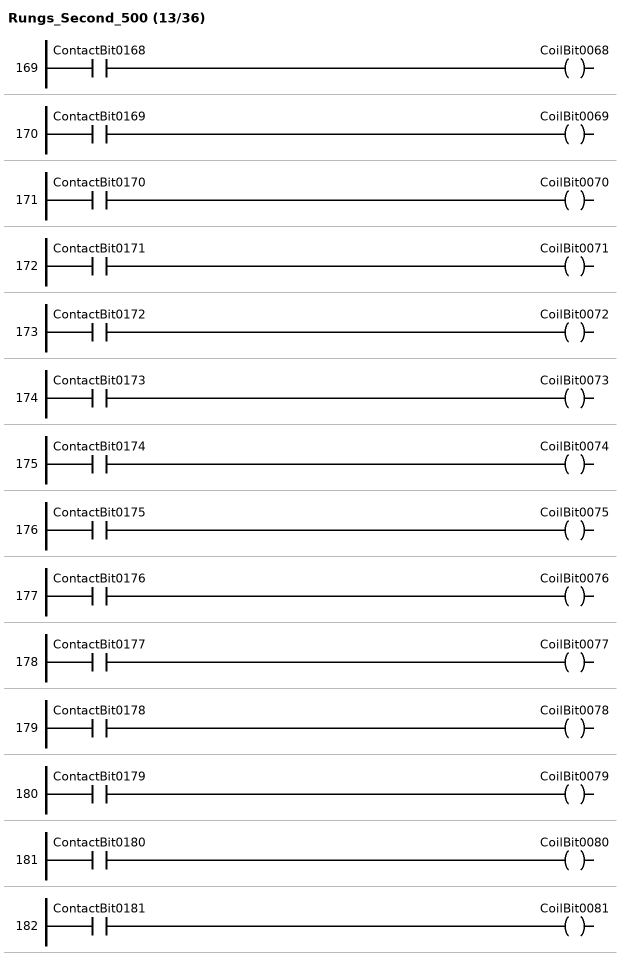
// NETWORK 169
CoilBit0068 := ContactBit0168;

// NETWORK 170
CoilBit0069 := ContactBit0169;

// NETWORK 171
CoilBit0070 := ContactBit0170;

// NETWORK 172
CoilBit0071 := ContactBit0171;

// NETWORK 173
CoilBit0072 := ContactBit0172;

// NETWORK 174
CoilBit0073 := ContactBit0173;

// NETWORK 175
CoilBit0074 := ContactBit0174;

// NETWORK 176
CoilBit0075 := ContactBit0175;

// NETWORK 177
CoilBit0076 := ContactBit0176;

// NETWORK 178
CoilBit0077 := ContactBit0177;

// NETWORK 179
CoilBit0078 := ContactBit0178;

// NETWORK 180
CoilBit0079 := ContactBit0179;

// NETWORK 181
CoilBit0080 := ContactBit0180;

// NETWORK 182
CoilBit0081 := ContactBit0181;

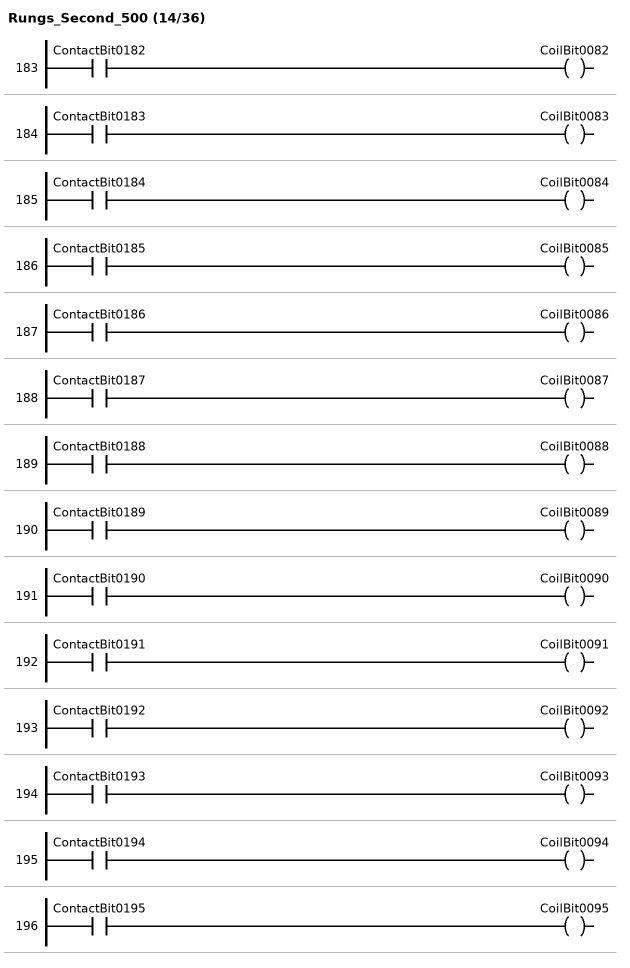
// NETWORK 183
CoilBit0082 := ContactBit0182;

// NETWORK 184
CoilBit0083 := ContactBit0183;

// NETWORK 185
CoilBit0084 := ContactBit0184;

// NETWORK 186
CoilBit0085 := ContactBit0185;

// NETWORK 187
CoilBit0086 := ContactBit0186;

// NETWORK 188
CoilBit0087 := ContactBit0187;

// NETWORK 189
CoilBit0088 := ContactBit0188;

// NETWORK 190
CoilBit0089 := ContactBit0189;

// NETWORK 191
CoilBit0090 := ContactBit0190;

// NETWORK 192
CoilBit0091 := ContactBit0191;

// NETWORK 193
CoilBit0092 := ContactBit0192;

// NETWORK 194
CoilBit0093 := ContactBit0193;

// NETWORK 195
CoilBit0094 := ContactBit0194;

// NETWORK 196
CoilBit0095 := ContactBit0195;

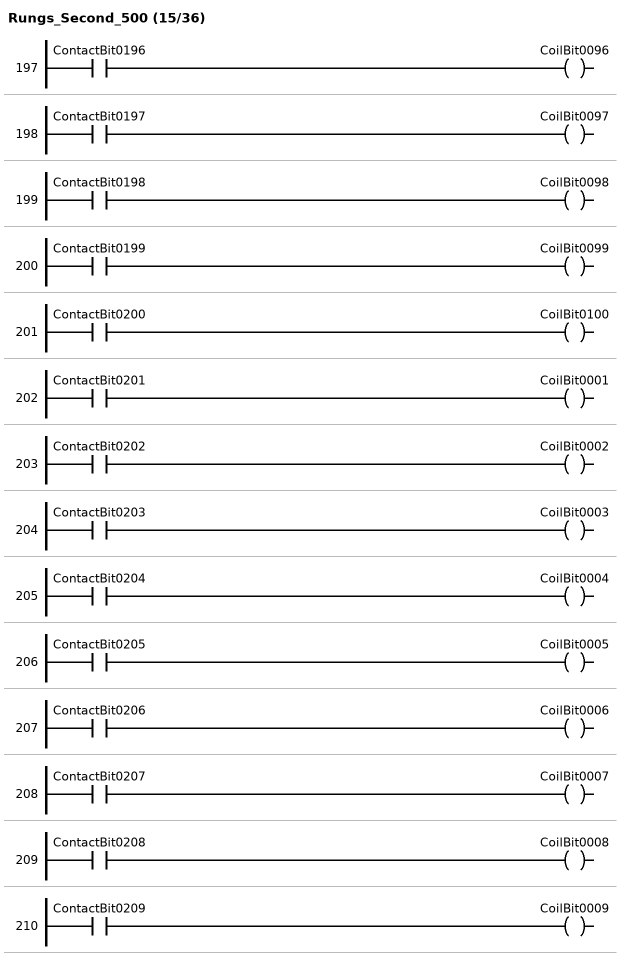
// NETWORK 197
CoilBit0096 := ContactBit0196;

// NETWORK 198
CoilBit0097 := ContactBit0197;

// NETWORK 199
CoilBit0098 := ContactBit0198;

// NETWORK 200
CoilBit0099 := ContactBit0199;

// NETWORK 201
CoilBit0100 := ContactBit0200;

// NETWORK 202
CoilBit0001 := ContactBit0201;

// NETWORK 203
CoilBit0002 := ContactBit0202;

// NETWORK 204
CoilBit0003 := ContactBit0203;

// NETWORK 205
CoilBit0004 := ContactBit0204;

// NETWORK 206
CoilBit0005 := ContactBit0205;

// NETWORK 207
CoilBit0006 := ContactBit0206;

// NETWORK 208
CoilBit0007 := ContactBit0207;

// NETWORK 209
CoilBit0008 := ContactBit0208;

// NETWORK 210
CoilBit0009 := ContactBit0209;

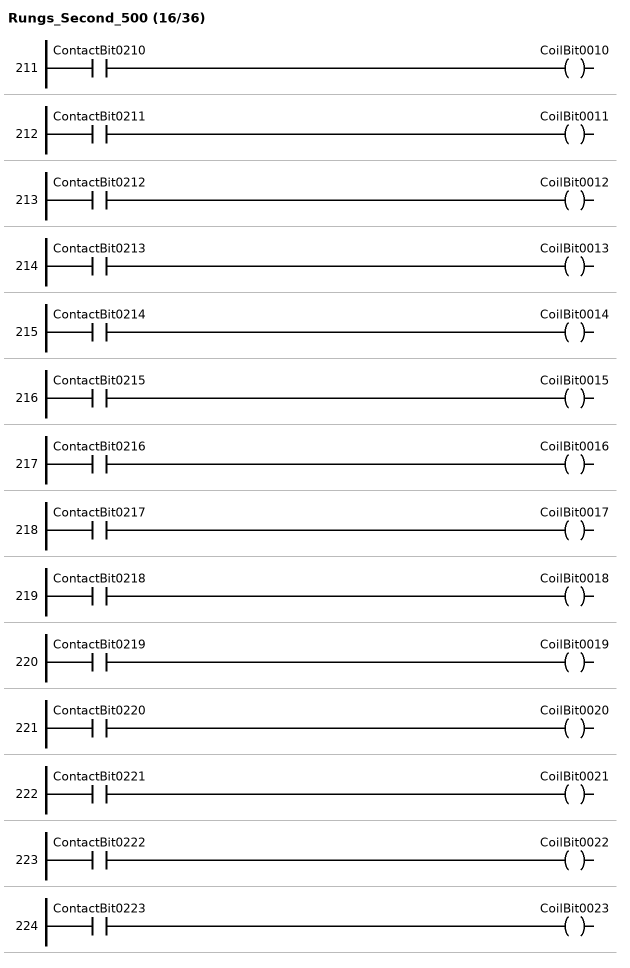
// NETWORK 211
CoilBit0010 := ContactBit0210;

// NETWORK 212
CoilBit0011 := ContactBit0211;

// NETWORK 213
CoilBit0012 := ContactBit0212;

// NETWORK 214
CoilBit0013 := ContactBit0213;

// NETWORK 215
CoilBit0014 := ContactBit0214;

// NETWORK 216
CoilBit0015 := ContactBit0215;

// NETWORK 217
CoilBit0016 := ContactBit0216;

// NETWORK 218
CoilBit0017 := ContactBit0217;

// NETWORK 219
CoilBit0018 := ContactBit0218;

// NETWORK 220
CoilBit0019 := ContactBit0219;

// NETWORK 221
CoilBit0020 := ContactBit0220;

// NETWORK 222
CoilBit0021 := ContactBit0221;

// NETWORK 223
CoilBit0022 := ContactBit0222;

// NETWORK 224
CoilBit0023 := ContactBit0223;

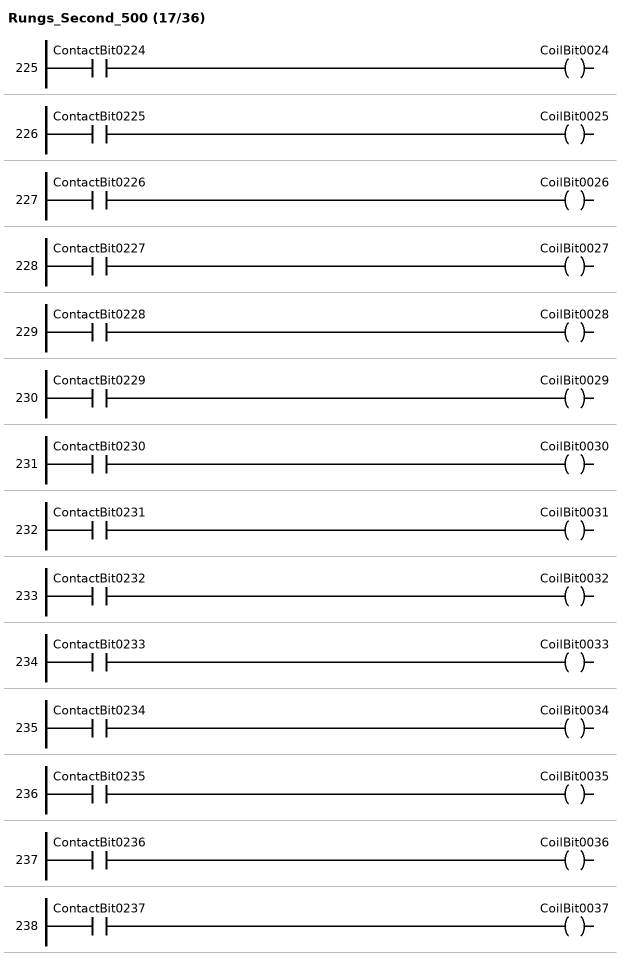
// NETWORK 225
CoilBit0024 := ContactBit0224;

// NETWORK 226
CoilBit0025 := ContactBit0225;

// NETWORK 227
CoilBit0026 := ContactBit0226;

// NETWORK 228
CoilBit0027 := ContactBit0227;

// NETWORK 229
CoilBit0028 := ContactBit0228;

// NETWORK 230
CoilBit0029 := ContactBit0229;

// NETWORK 231
CoilBit0030 := ContactBit0230;

// NETWORK 232
CoilBit0031 := ContactBit0231;

// NETWORK 233
CoilBit0032 := ContactBit0232;

// NETWORK 234
CoilBit0033 := ContactBit0233;

// NETWORK 235
CoilBit0034 := ContactBit0234;

// NETWORK 236
CoilBit0035 := ContactBit0235;

// NETWORK 237
CoilBit0036 := ContactBit0236;

// NETWORK 238
CoilBit0037 := ContactBit0237;

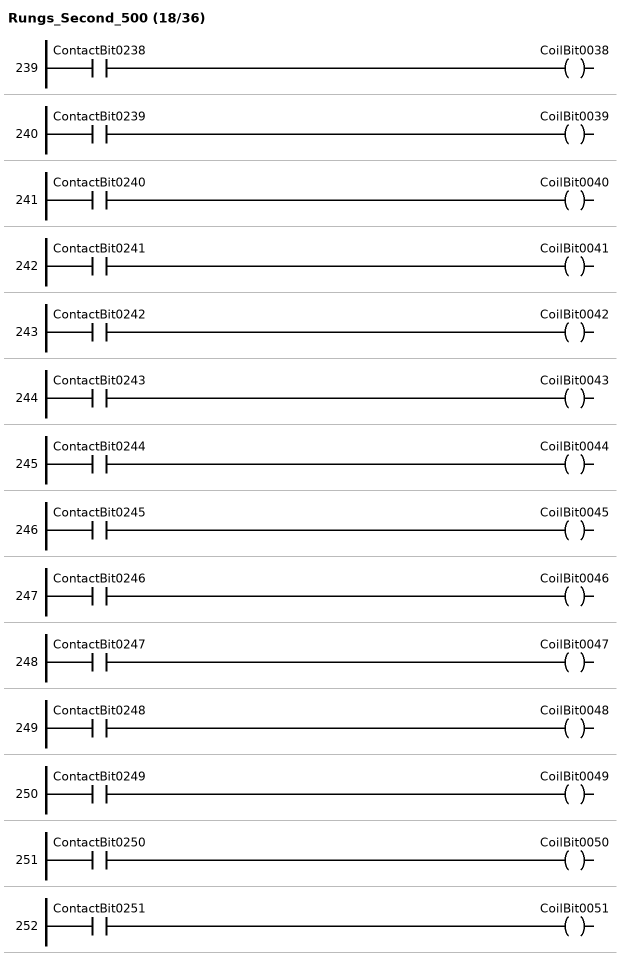
// NETWORK 239
CoilBit0038 := ContactBit0238;

// NETWORK 240
CoilBit0039 := ContactBit0239;

// NETWORK 241
CoilBit0040 := ContactBit0240;

// NETWORK 242
CoilBit0041 := ContactBit0241;

// NETWORK 243
CoilBit0042 := ContactBit0242;

// NETWORK 244
CoilBit0043 := ContactBit0243;

// NETWORK 245
CoilBit0044 := ContactBit0244;

// NETWORK 246
CoilBit0045 := ContactBit0245;

// NETWORK 247
CoilBit0046 := ContactBit0246;

// NETWORK 248
CoilBit0047 := ContactBit0247;

// NETWORK 249
CoilBit0048 := ContactBit0248;

// NETWORK 250
CoilBit0049 := ContactBit0249;

// NETWORK 251
CoilBit0050 := ContactBit0250;

// NETWORK 252
CoilBit0051 := ContactBit0251;

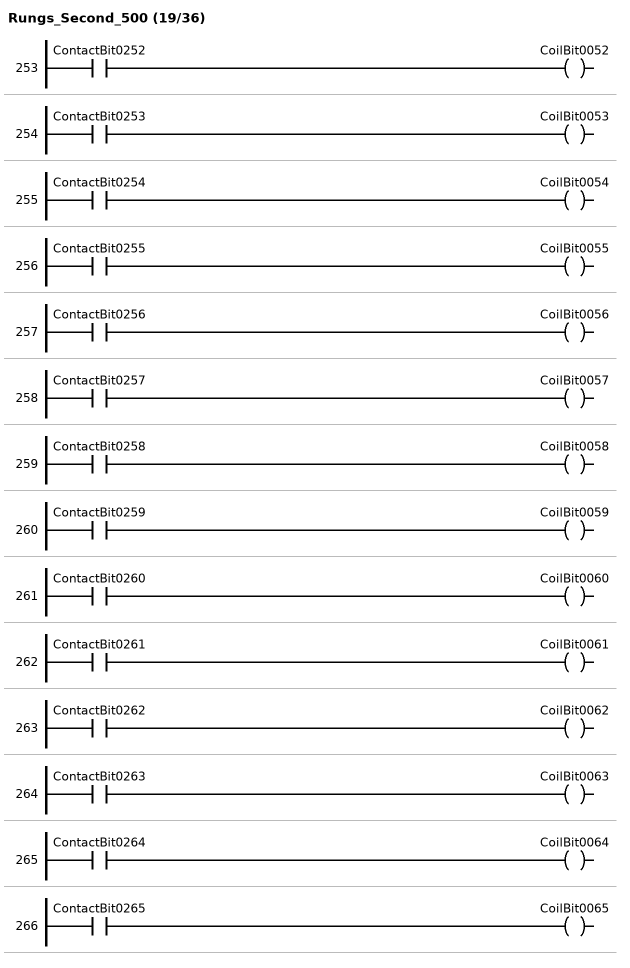
// NETWORK 253
CoilBit0052 := ContactBit0252;

// NETWORK 254
CoilBit0053 := ContactBit0253;

// NETWORK 255
CoilBit0054 := ContactBit0254;

// NETWORK 256
CoilBit0055 := ContactBit0255;

// NETWORK 257
CoilBit0056 := ContactBit0256;

// NETWORK 258
CoilBit0057 := ContactBit0257;

// NETWORK 259
CoilBit0058 := ContactBit0258;

// NETWORK 260
CoilBit0059 := ContactBit0259;

// NETWORK 261
CoilBit0060 := ContactBit0260;

// NETWORK 262
CoilBit0061 := ContactBit0261;

// NETWORK 263
CoilBit0062 := ContactBit0262;

// NETWORK 264
CoilBit0063 := ContactBit0263;

// NETWORK 265
CoilBit0064 := ContactBit0264;

// NETWORK 266
CoilBit0065 := ContactBit0265;

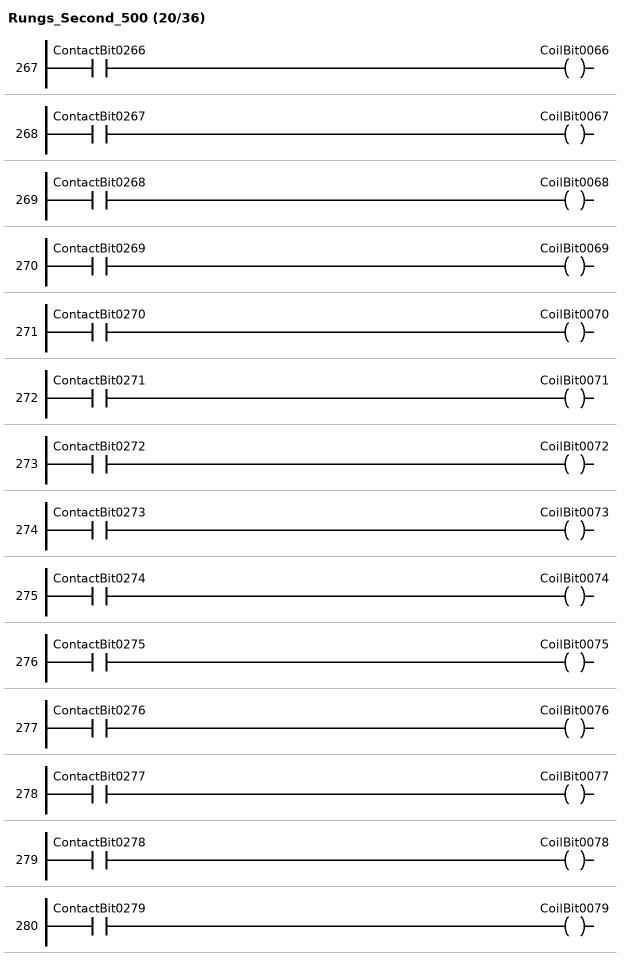
// NETWORK 267
CoilBit0066 := ContactBit0266;

// NETWORK 268
CoilBit0067 := ContactBit0267;

// NETWORK 269
CoilBit0068 := ContactBit0268;

// NETWORK 270
CoilBit0069 := ContactBit0269;

// NETWORK 271
CoilBit0070 := ContactBit0270;

// NETWORK 272
CoilBit0071 := ContactBit0271;

// NETWORK 273
CoilBit0072 := ContactBit0272;

// NETWORK 274
CoilBit0073 := ContactBit0273;

// NETWORK 275
CoilBit0074 := ContactBit0274;

// NETWORK 276
CoilBit0075 := ContactBit0275;

// NETWORK 277
CoilBit0076 := ContactBit0276;

// NETWORK 278
CoilBit0077 := ContactBit0277;

// NETWORK 279
CoilBit0078 := ContactBit0278;

// NETWORK 280
CoilBit0079 := ContactBit0279;

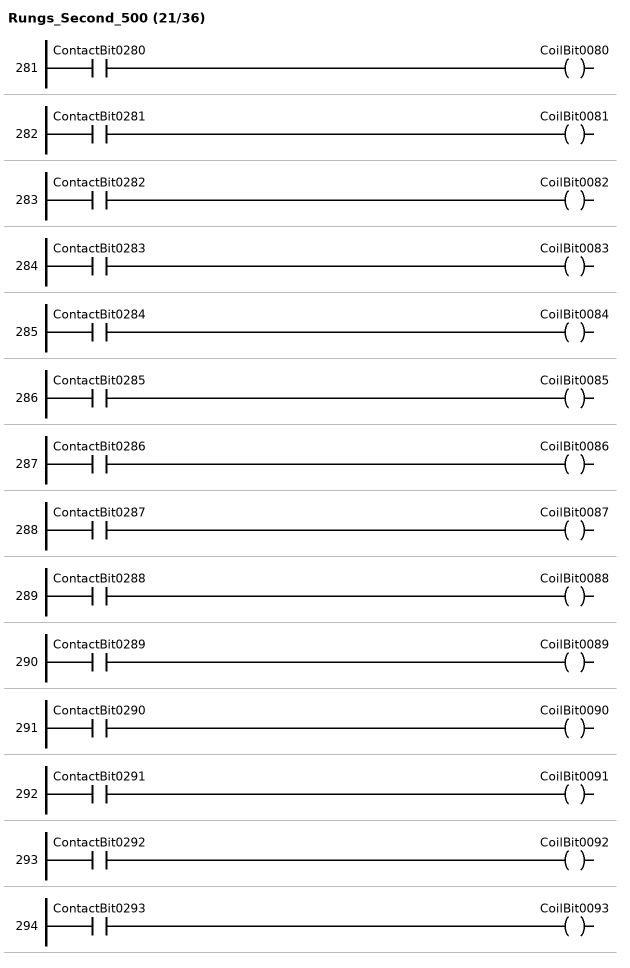
// NETWORK 281
CoilBit0080 := ContactBit0280;

// NETWORK 282
CoilBit0081 := ContactBit0281;

// NETWORK 283
CoilBit0082 := ContactBit0282;

// NETWORK 284
CoilBit0083 := ContactBit0283;

// NETWORK 285
CoilBit0084 := ContactBit0284;

// NETWORK 286
CoilBit0085 := ContactBit0285;

// NETWORK 287
CoilBit0086 := ContactBit0286;

// NETWORK 288
CoilBit0087 := ContactBit0287;

// NETWORK 289
CoilBit0088 := ContactBit0288;

// NETWORK 290
CoilBit0089 := ContactBit0289;

// NETWORK 291
CoilBit0090 := ContactBit0290;

// NETWORK 292
CoilBit0091 := ContactBit0291;

// NETWORK 293
CoilBit0092 := ContactBit0292;

// NETWORK 294
CoilBit0093 := ContactBit0293;

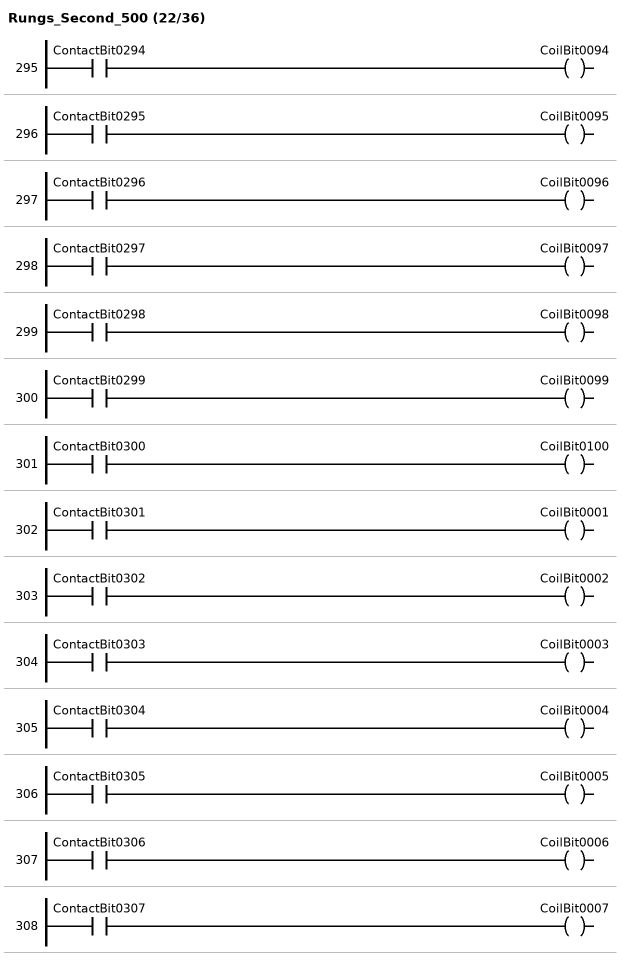
// NETWORK 295
CoilBit0094 := ContactBit0294;

// NETWORK 296
CoilBit0095 := ContactBit0295;

// NETWORK 297
CoilBit0096 := ContactBit0296;

// NETWORK 298
CoilBit0097 := ContactBit0297;

// NETWORK 299
CoilBit0098 := ContactBit0298;

// NETWORK 300
CoilBit0099 := ContactBit0299;

// NETWORK 301
CoilBit0100 := ContactBit0300;

// NETWORK 302
CoilBit0001 := ContactBit0301;

// NETWORK 303
CoilBit0002 := ContactBit0302;

// NETWORK 304
CoilBit0003 := ContactBit0303;

// NETWORK 305
CoilBit0004 := ContactBit0304;

// NETWORK 306
CoilBit0005 := ContactBit0305;

// NETWORK 307
CoilBit0006 := ContactBit0306;

// NETWORK 308
CoilBit0007 := ContactBit0307;

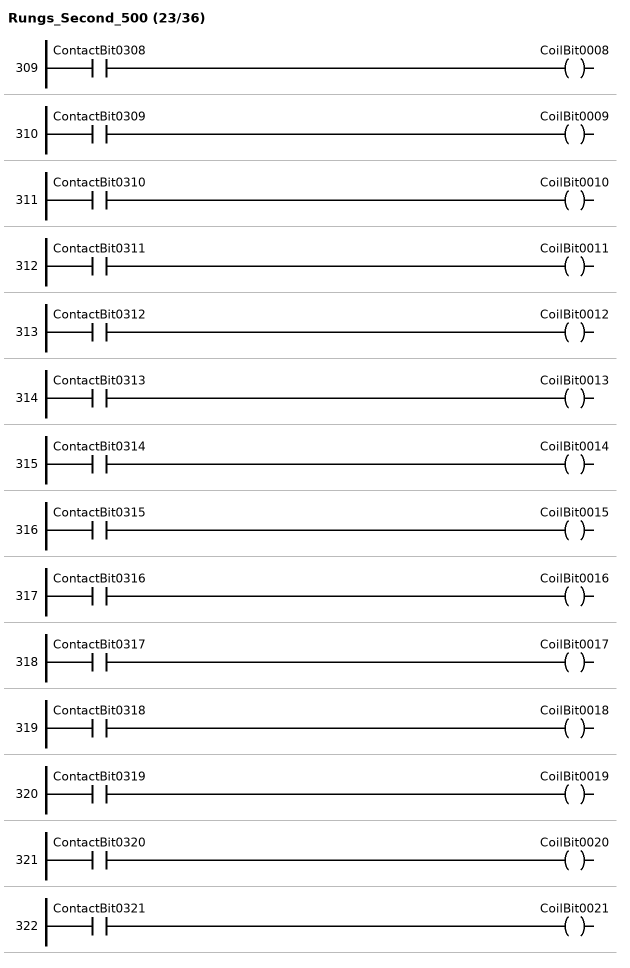
// NETWORK 309
CoilBit0008 := ContactBit0308;

// NETWORK 310
CoilBit0009 := ContactBit0309;

// NETWORK 311
CoilBit0010 := ContactBit0310;

// NETWORK 312
CoilBit0011 := ContactBit0311;

// NETWORK 313
CoilBit0012 := ContactBit0312;

// NETWORK 314
CoilBit0013 := ContactBit0313;

// NETWORK 315
CoilBit0014 := ContactBit0314;

// NETWORK 316
CoilBit0015 := ContactBit0315;

// NETWORK 317
CoilBit0016 := ContactBit0316;

// NETWORK 318
CoilBit0017 := ContactBit0317;

// NETWORK 319
CoilBit0018 := ContactBit0318;

// NETWORK 320
CoilBit0019 := ContactBit0319;

// NETWORK 321
CoilBit0020 := ContactBit0320;

// NETWORK 322
CoilBit0021 := ContactBit0321;

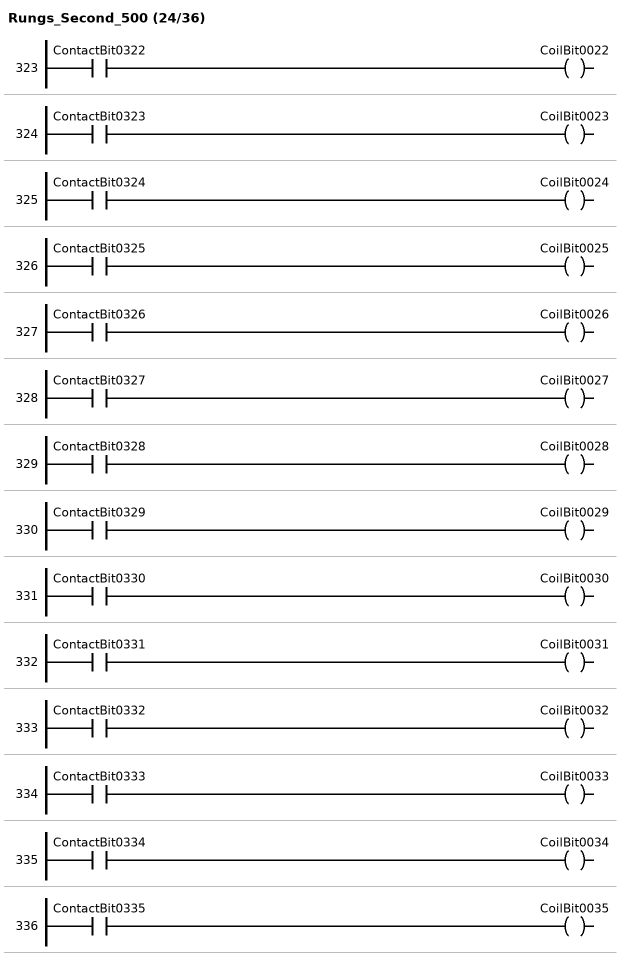
// NETWORK 323
CoilBit0022 := ContactBit0322;

// NETWORK 324
CoilBit0023 := ContactBit0323;

// NETWORK 325
CoilBit0024 := ContactBit0324;

// NETWORK 326
CoilBit0025 := ContactBit0325;

// NETWORK 327
CoilBit0026 := ContactBit0326;

// NETWORK 328
CoilBit0027 := ContactBit0327;

// NETWORK 329
CoilBit0028 := ContactBit0328;

// NETWORK 330
CoilBit0029 := ContactBit0329;

// NETWORK 331
CoilBit0030 := ContactBit0330;

// NETWORK 332
CoilBit0031 := ContactBit0331;

// NETWORK 333
CoilBit0032 := ContactBit0332;

// NETWORK 334
CoilBit0033 := ContactBit0333;

// NETWORK 335
CoilBit0034 := ContactBit0334;

// NETWORK 336
CoilBit0035 := ContactBit0335;

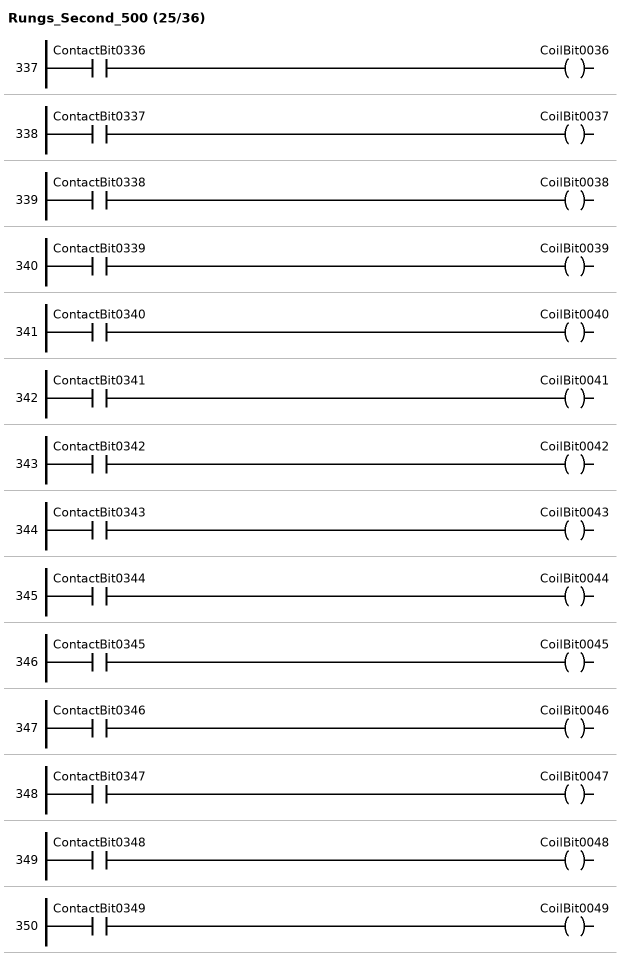
// NETWORK 337
CoilBit0036 := ContactBit0336;

// NETWORK 338
CoilBit0037 := ContactBit0337;

// NETWORK 339
CoilBit0038 := ContactBit0338;

// NETWORK 340
CoilBit0039 := ContactBit0339;

// NETWORK 341
CoilBit0040 := ContactBit0340;

// NETWORK 342
CoilBit0041 := ContactBit0341;

// NETWORK 343
CoilBit0042 := ContactBit0342;

// NETWORK 344
CoilBit0043 := ContactBit0343;

// NETWORK 345
CoilBit0044 := ContactBit0344;

// NETWORK 346
CoilBit0045 := ContactBit0345;

// NETWORK 347
CoilBit0046 := ContactBit0346;

// NETWORK 348
CoilBit0047 := ContactBit0347;

// NETWORK 349
CoilBit0048 := ContactBit0348;

// NETWORK 350
CoilBit0049 := ContactBit0349;

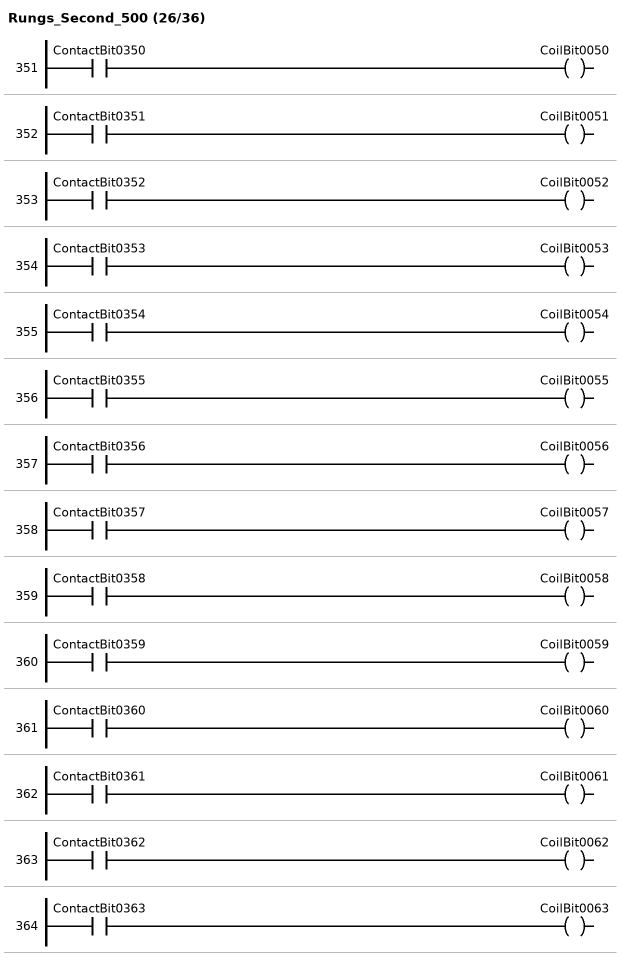
// NETWORK 351
CoilBit0050 := ContactBit0350;

// NETWORK 352
CoilBit0051 := ContactBit0351;

// NETWORK 353
CoilBit0052 := ContactBit0352;

// NETWORK 354
CoilBit0053 := ContactBit0353;

// NETWORK 355
CoilBit0054 := ContactBit0354;

// NETWORK 356
CoilBit0055 := ContactBit0355;

// NETWORK 357
CoilBit0056 := ContactBit0356;

// NETWORK 358
CoilBit0057 := ContactBit0357;

// NETWORK 359
CoilBit0058 := ContactBit0358;

// NETWORK 360
CoilBit0059 := ContactBit0359;

// NETWORK 361
CoilBit0060 := ContactBit0360;

// NETWORK 362
CoilBit0061 := ContactBit0361;

// NETWORK 363
CoilBit0062 := ContactBit0362;

// NETWORK 364
CoilBit0063 := ContactBit0363;

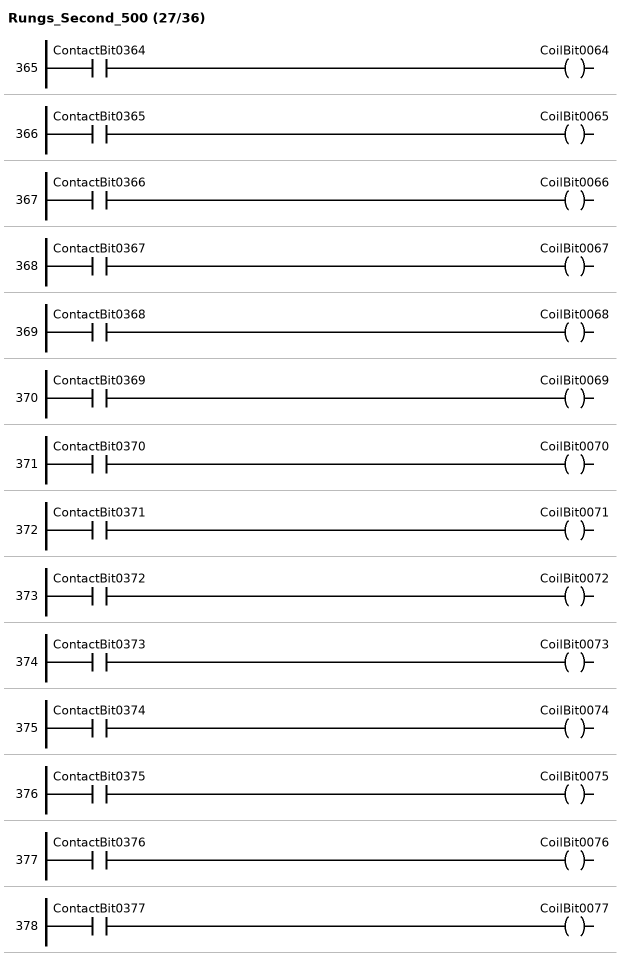
// NETWORK 365
CoilBit0064 := ContactBit0364;

// NETWORK 366
CoilBit0065 := ContactBit0365;

// NETWORK 367
CoilBit0066 := ContactBit0366;

// NETWORK 368
CoilBit0067 := ContactBit0367;

// NETWORK 369
CoilBit0068 := ContactBit0368;

// NETWORK 370
CoilBit0069 := ContactBit0369;

// NETWORK 371
CoilBit0070 := ContactBit0370;

// NETWORK 372
CoilBit0071 := ContactBit0371;

// NETWORK 373
CoilBit0072 := ContactBit0372;

// NETWORK 374
CoilBit0073 := ContactBit0373;

// NETWORK 375
CoilBit0074 := ContactBit0374;

// NETWORK 376
CoilBit0075 := ContactBit0375;

// NETWORK 377
CoilBit0076 := ContactBit0376;

// NETWORK 378
CoilBit0077 := ContactBit0377;

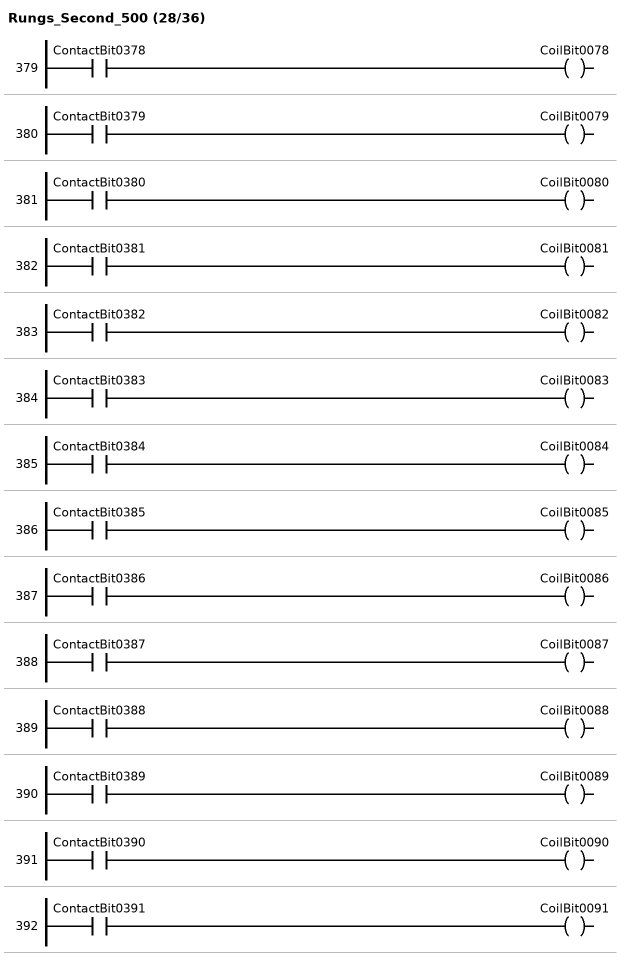
// NETWORK 379
CoilBit0078 := ContactBit0378;

// NETWORK 380
CoilBit0079 := ContactBit0379;

// NETWORK 381
CoilBit0080 := ContactBit0380;

// NETWORK 382
CoilBit0081 := ContactBit0381;

// NETWORK 383
CoilBit0082 := ContactBit0382;

// NETWORK 384
CoilBit0083 := ContactBit0383;

// NETWORK 385
CoilBit0084 := ContactBit0384;

// NETWORK 386
CoilBit0085 := ContactBit0385;

// NETWORK 387
CoilBit0086 := ContactBit0386;

// NETWORK 388
CoilBit0087 := ContactBit0387;

// NETWORK 389
CoilBit0088 := ContactBit0388;

// NETWORK 390
CoilBit0089 := ContactBit0389;

// NETWORK 391
CoilBit0090 := ContactBit0390;

// NETWORK 392
CoilBit0091 := ContactBit0391;

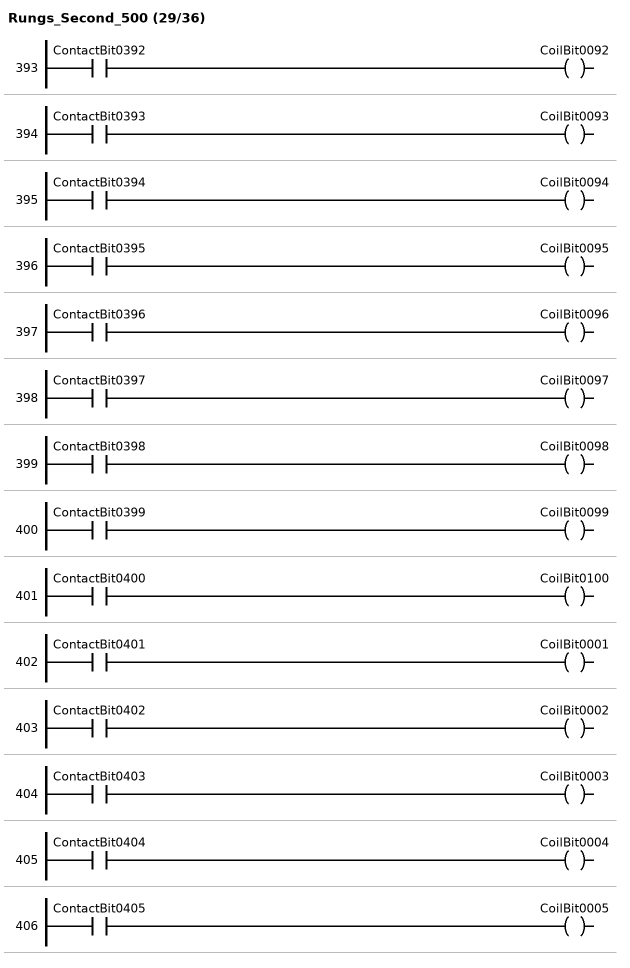
// NETWORK 393
CoilBit0092 := ContactBit0392;

// NETWORK 394
CoilBit0093 := ContactBit0393;

// NETWORK 395
CoilBit0094 := ContactBit0394;

// NETWORK 396
CoilBit0095 := ContactBit0395;

// NETWORK 397
CoilBit0096 := ContactBit0396;

// NETWORK 398
CoilBit0097 := ContactBit0397;

// NETWORK 399
CoilBit0098 := ContactBit0398;

// NETWORK 400
CoilBit0099 := ContactBit0399;

// NETWORK 401
CoilBit0100 := ContactBit0400;

// NETWORK 402
CoilBit0001 := ContactBit0401;

// NETWORK 403
CoilBit0002 := ContactBit0402;

// NETWORK 404
CoilBit0003 := ContactBit0403;

// NETWORK 405
CoilBit0004 := ContactBit0404;

// NETWORK 406
CoilBit0005 := ContactBit0405;

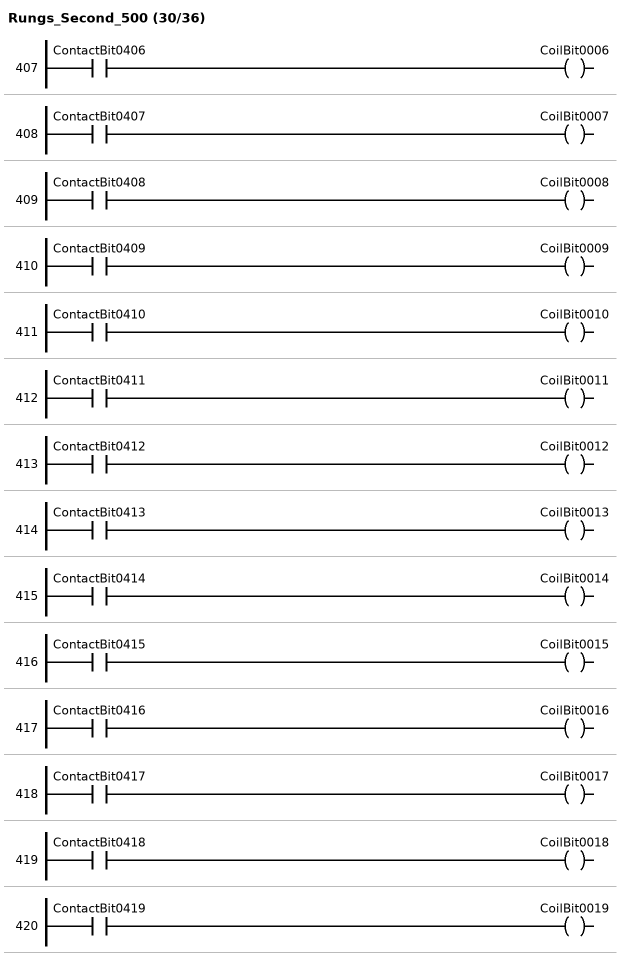
// NETWORK 407
CoilBit0006 := ContactBit0406;

// NETWORK 408
CoilBit0007 := ContactBit0407;

// NETWORK 409
CoilBit0008 := ContactBit0408;

// NETWORK 410
CoilBit0009 := ContactBit0409;

// NETWORK 411
CoilBit0010 := ContactBit0410;

// NETWORK 412
CoilBit0011 := ContactBit0411;

// NETWORK 413
CoilBit0012 := ContactBit0412;

// NETWORK 414
CoilBit0013 := ContactBit0413;

// NETWORK 415
CoilBit0014 := ContactBit0414;

// NETWORK 416
CoilBit0015 := ContactBit0415;

// NETWORK 417
CoilBit0016 := ContactBit0416;

// NETWORK 418
CoilBit0017 := ContactBit0417;

// NETWORK 419
CoilBit0018 := ContactBit0418;

// NETWORK 420
CoilBit0019 := ContactBit0419;

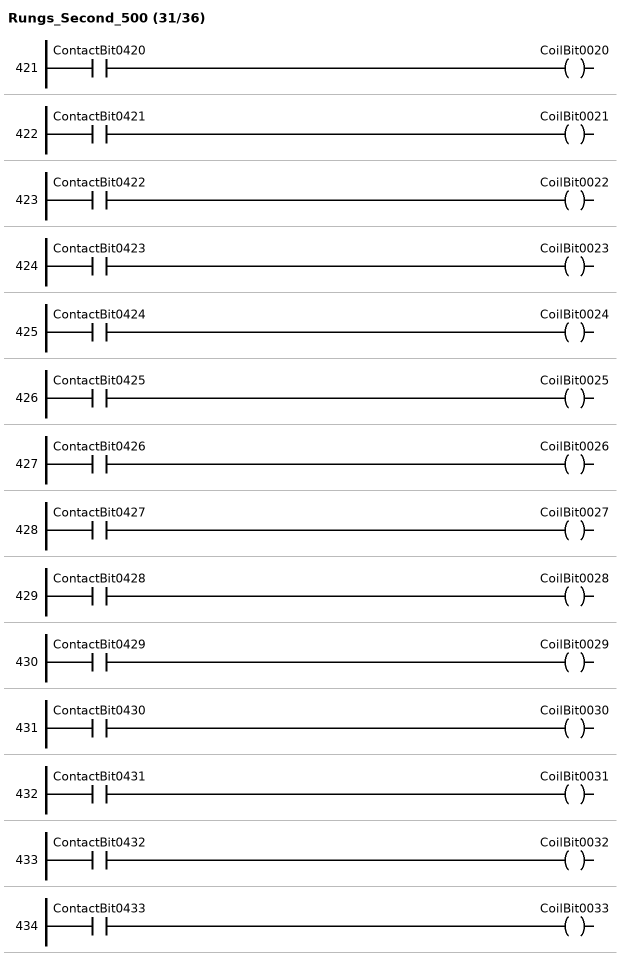
// NETWORK 421
CoilBit0020 := ContactBit0420;

// NETWORK 422
CoilBit0021 := ContactBit0421;

// NETWORK 423
CoilBit0022 := ContactBit0422;

// NETWORK 424
CoilBit0023 := ContactBit0423;

// NETWORK 425
CoilBit0024 := ContactBit0424;

// NETWORK 426
CoilBit0025 := ContactBit0425;

// NETWORK 427
CoilBit0026 := ContactBit0426;

// NETWORK 428
CoilBit0027 := ContactBit0427;

// NETWORK 429
CoilBit0028 := ContactBit0428;

// NETWORK 430
CoilBit0029 := ContactBit0429;

// NETWORK 431
CoilBit0030 := ContactBit0430;

// NETWORK 432
CoilBit0031 := ContactBit0431;

// NETWORK 433
CoilBit0032 := ContactBit0432;

// NETWORK 434
CoilBit0033 := ContactBit0433;

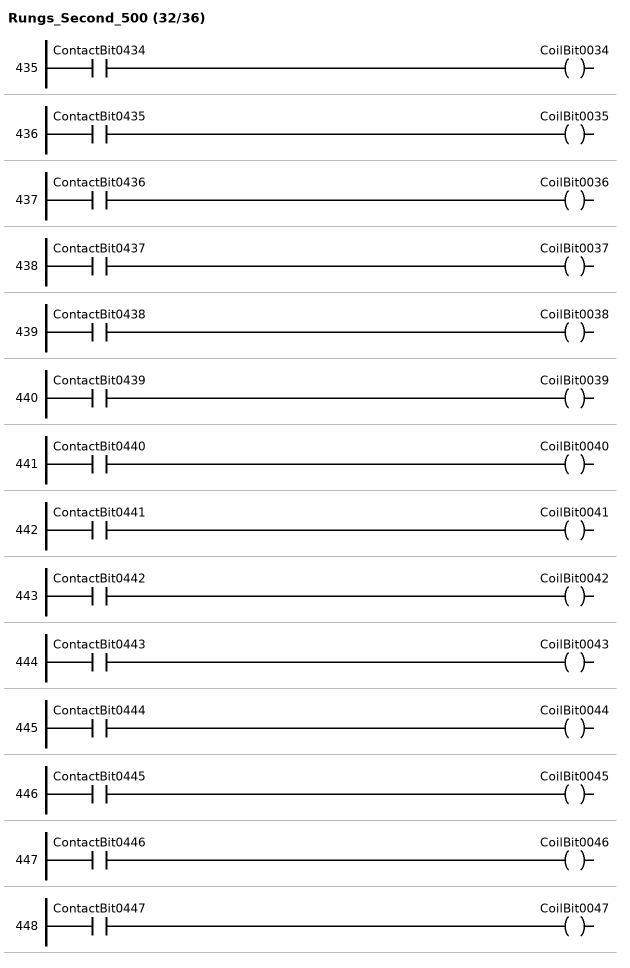
// NETWORK 435
CoilBit0034 := ContactBit0434;

// NETWORK 436
CoilBit0035 := ContactBit0435;

// NETWORK 437
CoilBit0036 := ContactBit0436;

// NETWORK 438
CoilBit0037 := ContactBit0437;

// NETWORK 439
CoilBit0038 := ContactBit0438;

// NETWORK 440
CoilBit0039 := ContactBit0439;

// NETWORK 441
CoilBit0040 := ContactBit0440;

// NETWORK 442
CoilBit0041 := ContactBit0441;

// NETWORK 443
CoilBit0042 := ContactBit0442;

// NETWORK 444
CoilBit0043 := ContactBit0443;

// NETWORK 445
CoilBit0044 := ContactBit0444;

// NETWORK 446
CoilBit0045 := ContactBit0445;

// NETWORK 447
CoilBit0046 := ContactBit0446;

// NETWORK 448
CoilBit0047 := ContactBit0447;

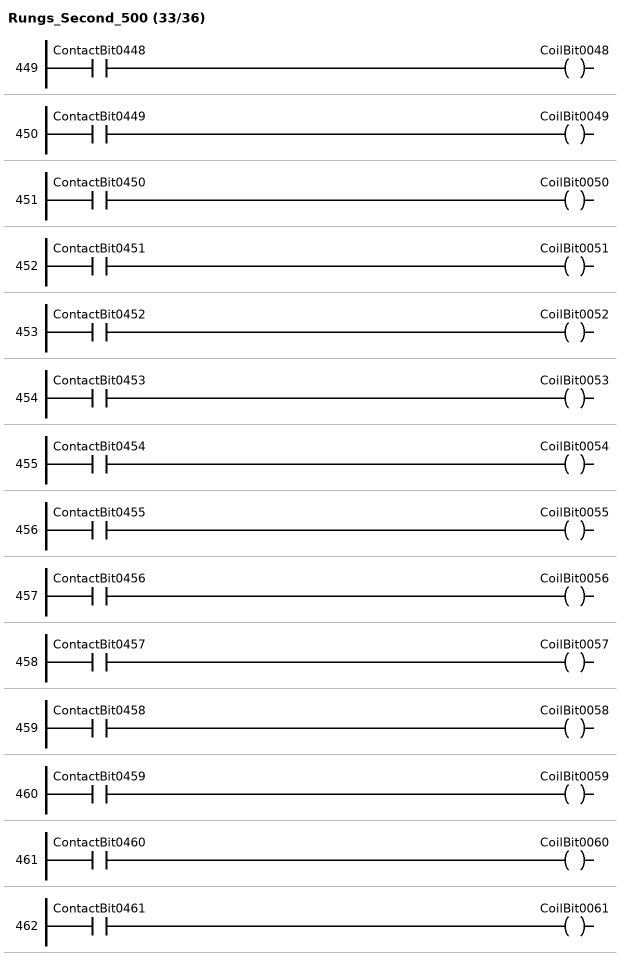
// NETWORK 449
CoilBit0048 := ContactBit0448;

// NETWORK 450
CoilBit0049 := ContactBit0449;

// NETWORK 451
CoilBit0050 := ContactBit0450;

// NETWORK 452
CoilBit0051 := ContactBit0451;

// NETWORK 453
CoilBit0052 := ContactBit0452;

// NETWORK 454
CoilBit0053 := ContactBit0453;

// NETWORK 455
CoilBit0054 := ContactBit0454;

// NETWORK 456
CoilBit0055 := ContactBit0455;

// NETWORK 457
CoilBit0056 := ContactBit0456;

// NETWORK 458
CoilBit0057 := ContactBit0457;

// NETWORK 459
CoilBit0058 := ContactBit0458;

// NETWORK 460
CoilBit0059 := ContactBit0459;

// NETWORK 461
CoilBit0060 := ContactBit0460;

// NETWORK 462
CoilBit0061 := ContactBit0461;

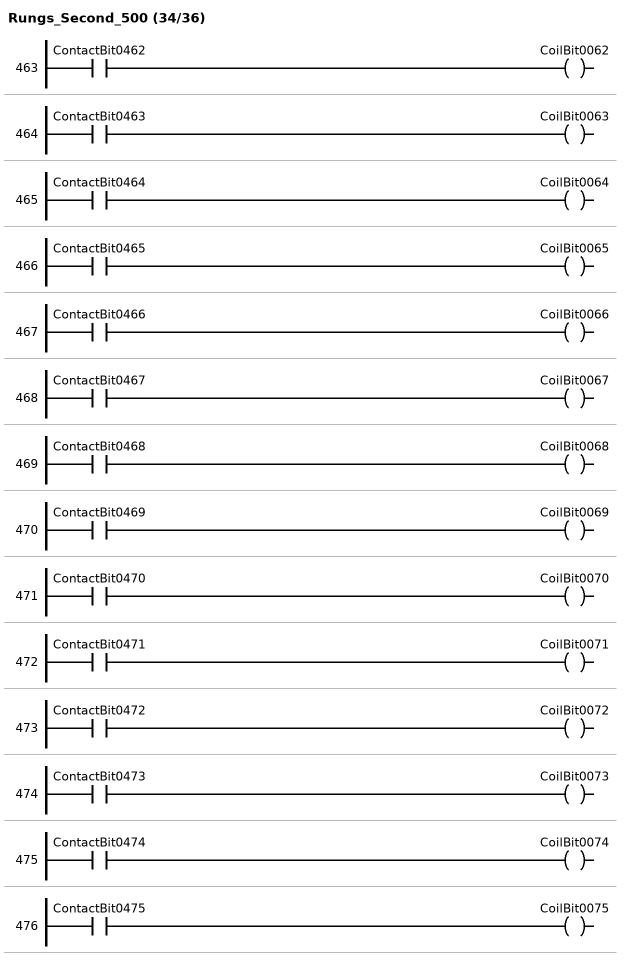
// NETWORK 463
CoilBit0062 := ContactBit0462;

// NETWORK 464
CoilBit0063 := ContactBit0463;

// NETWORK 465
CoilBit0064 := ContactBit0464;

// NETWORK 466
CoilBit0065 := ContactBit0465;

// NETWORK 467
CoilBit0066 := ContactBit0466;

// NETWORK 468
CoilBit0067 := ContactBit0467;

// NETWORK 469
CoilBit0068 := ContactBit0468;

// NETWORK 470
CoilBit0069 := ContactBit0469;

// NETWORK 471
CoilBit0070 := ContactBit0470;

// NETWORK 472
CoilBit0071 := ContactBit0471;

// NETWORK 473
CoilBit0072 := ContactBit0472;

// NETWORK 474
CoilBit0073 := ContactBit0473;

// NETWORK 475
CoilBit0074 := ContactBit0474;

// NETWORK 476
CoilBit0075 := ContactBit0475;

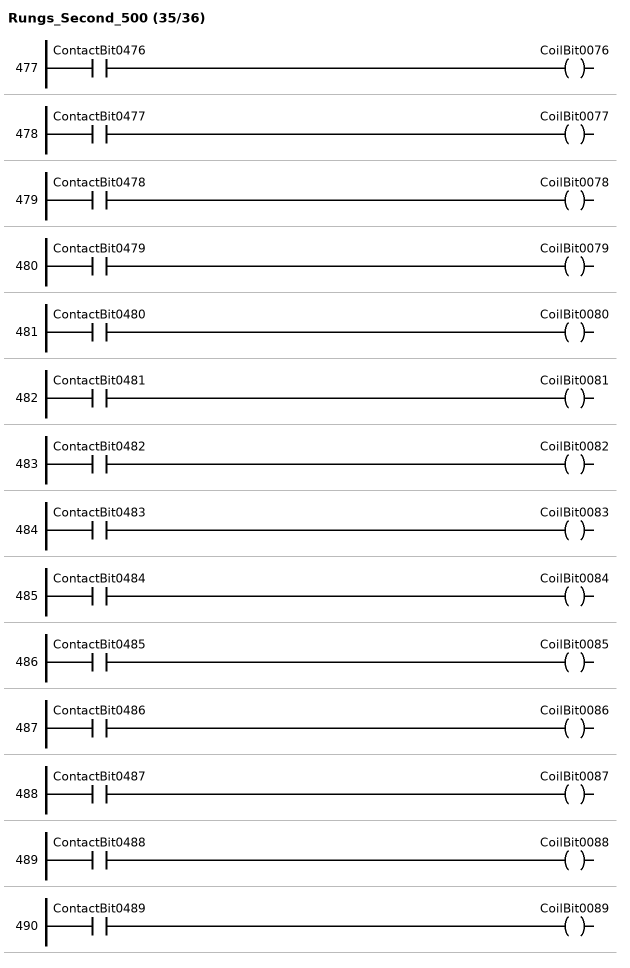
// NETWORK 477
CoilBit0076 := ContactBit0476;

// NETWORK 478
CoilBit0077 := ContactBit0477;

// NETWORK 479
CoilBit0078 := ContactBit0478;

// NETWORK 480
CoilBit0079 := ContactBit0479;

// NETWORK 481
CoilBit0080 := ContactBit0480;

// NETWORK 482
CoilBit0081 := ContactBit0481;

// NETWORK 483
CoilBit0082 := ContactBit0482;

// NETWORK 484
CoilBit0083 := ContactBit0483;

// NETWORK 485
CoilBit0084 := ContactBit0484;

// NETWORK 486
CoilBit0085 := ContactBit0485;

// NETWORK 487
CoilBit0086 := ContactBit0486;

// NETWORK 488
CoilBit0087 := ContactBit0487;

// NETWORK 489
CoilBit0088 := ContactBit0488;

// NETWORK 490
CoilBit0089 := ContactBit0489;

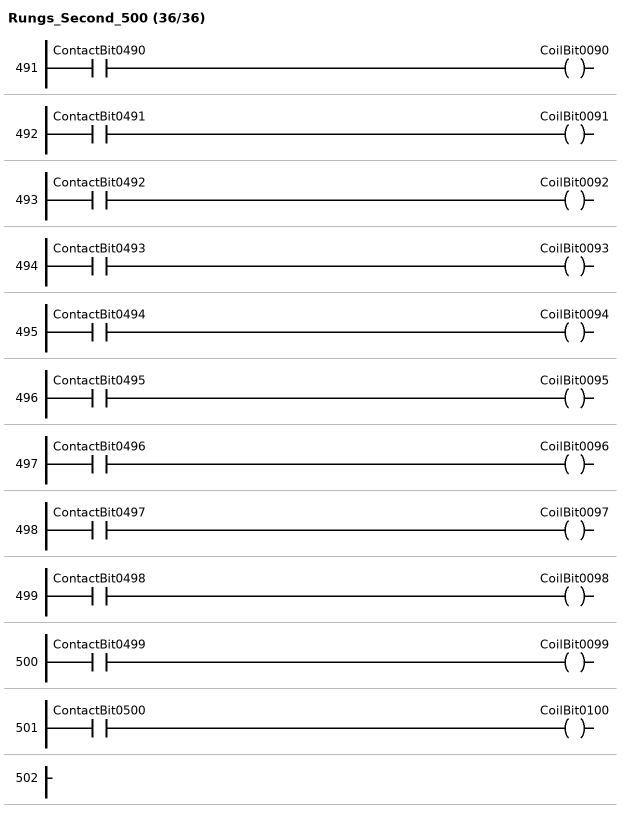
// NETWORK 491
CoilBit0090 := ContactBit0490;

// NETWORK 492
CoilBit0091 := ContactBit0491;

// NETWORK 493
CoilBit0092 := ContactBit0492;

// NETWORK 494
CoilBit0093 := ContactBit0493;

// NETWORK 495
CoilBit0094 := ContactBit0494;

// NETWORK 496
CoilBit0095 := ContactBit0495;

// NETWORK 497
CoilBit0096 := ContactBit0496;

// NETWORK 498
CoilBit0097 := ContactBit0497;

// NETWORK 499
CoilBit0098 := ContactBit0498;

// NETWORK 500
CoilBit0099 := ContactBit0499;

// NETWORK 501
CoilBit0100 := ContactBit0500;

// NETWORK 502

END_PROGRAM

// RunMotion_All
PROGRAM RunMotion_All
VAR
	DoMotion_X: MotionFB;
	DoMotion_Y: MotionFB;
	DoMotion_Z: MotionFB;
	DoMotion_A: MotionFB;
	DoMotion_B: MotionFB;
	
END_VAR

DoMotion_X(AxisVar:=X, Enable:=TRUE);
DoMotion_Y(AxisVar:=Y, Enable:=TRUE);
DoMotion_Z(AxisVar:=Z, Enable:=TRUE);
DoMotion_A(AxisVar:=A, Enable:=TRUE);
DoMotion_B(AxisVar:=ZZ, Enable:=TRUE);

END_PROGRAM

// MotionFB
FUNCTION_BLOCK MotionFB
VAR_IN_OUT
	AxisVar: AXIS_REF_SM3;
END_VAR
VAR_INPUT
	Enable:BOOL;
END_VAR
VAR_OUTPUT
	Running:BOOL;
END_VAR
VAR
		AxisControl : IO_AxisControl;
	iStatus: INT := -2;
	DoMove : MC_MoveRelative;
	TimerON:TON;
	tWait : TIME := T#5S;
	tWaitPowerup: TIME := T#30S;
	Got_DC_OutOfSync: BOOL;

	Restart_Axis : SMC3_ReinitDrive;
	TimerRecover : TON;
	EnableAxisControl : BOOL := FALSE;
	
	
	HMI_ActualPosition: INT;
	ActualPosition: LREAL;
END_VAR

IF Enable = FALSE THEN
(*	
	IF AxisVar.nAxisState <> standstill THEN
		In_Stop:= TRUE;
	END_IF
*)	
	Running:= FALSE;
	RETURN;
ELSE
	Running:= True;
//	In_Stop := FALSE;
END_IF

IF iStatus > -1 AND NOT(DC_InSync) THEN
	Got_DC_OutOfSync := TRUE;
	(* //Commented Out to use Recovery
	iStatus := 10; 
	gSyncErrors := gSyncErrors + 1
	*)
END_IF

CASE iStatus OF
	
-2: //Wait Time
	EnableAxisControl:= FALSE;
	//TimerON(PT:=tWaitPowerup, IN:=TRUE);
	IF EtherCAT_Master.xConfigFinished AND DC_InSync THEN
		//TimerON(IN:=FALSE,PT:=T#0S);
		iStatus:=iStatus + 1;
	END_IF
	
-1: //Wait Time
	EnableAxisControl:=TRUE;
	IF DC_InSync THEN
		iStatus:=iStatus + 1;
	END_IF
	
	
0: //Wait for Drive to be ready
	//AxisControl(Axis:=X, Enable:=TRUE);
	//In_Power:=TRUE;
	IF AxisControl.Ready AND AxisVar.nAxisState=standstill THEN
		IF In_Cycle = TRUE THEN
			iStatus:=iStatus + 1;
		ELSE
			iStatus:=0;	
		END_IF
	END_IF;
	
1: //Start positive move
	DoMove(Axis:=AxisVar, Distance:= g_PosDistance, Velocity:=g_Vel, Acceleration:=g_Acc, Deceleration:=g_Acc, Execute:= TRUE);
	IF DoMove.Busy THEN 
		IF In_Cycle = TRUE THEN
			iStatus:=iStatus + 1;
		ELSE
			iStatus:=0;	
		END_IF
	END_IF
	
2: // Wait for Move Finish
	DoMove(Axis:=AxisVar, Distance:= g_PosDistance, Velocity:=g_Vel, Acceleration:=g_Acc, Deceleration:=g_Acc, Execute:= TRUE);
	IF DoMove.Done AND AxisVar.nAxisState=standstill THEN 
		DoMove(Axis:=AxisVar, Execute:= FALSE);
		
		IF In_Cycle = TRUE THEN
			iStatus:=iStatus + 1;
		ELSE
			iStatus:=0;	
		END_IF
	END_IF
	
3: //Wait Time
	g_MoveDwellPos := TRUE;
	TimerON(PT:=tWait, IN:=TRUE);
	IF TimerON.Q=TRUE THEN
		TimerON(IN:=FALSE,PT:=T#0S);
		g_MoveDwellPos :=  FALSE;
		IF In_Cycle = TRUE THEN
			iStatus:=iStatus + 1;
		ELSE
			iStatus:=0;	
		END_IF
	END_IF

4: //Start negative move
	DoMove(Axis:=AxisVar, Distance:= g_NegDistance, Velocity:=g_Vel, Acceleration:=g_Acc, Deceleration:=g_Acc, Execute:= TRUE);
	IF DoMove.Busy THEN 
		IF In_Cycle = TRUE THEN
			iStatus:=iStatus + 1;
		ELSE
			iStatus:=0;	
		END_IF
	END_IF
	
5: // Wait for Move Finish
	DoMove(Axis:=AxisVar, Distance:= g_NegDistance, Velocity:=g_Vel, Acceleration:=g_Acc, Deceleration:=g_Acc, Execute:= TRUE);
	IF DoMove.Done AND AxisVar.nAxisState=standstill THEN 
		DoMove(Axis:=AxisVar, Execute:= FALSE);
		IF In_Cycle = TRUE THEN
			iStatus:=iStatus + 1;
		ELSE
			iStatus:=0;	
		END_IF
	END_IF
	
6: //Wait Time
	g_MoveDwellNeg := TRUE;
	TimerON(PT:=tWait, IN:=TRUE);
	IF TimerON.Q=TRUE THEN
		TimerON(IN:=FALSE,PT:=T#0S);
		iStatus:=0;
		g_MoveDwellNeg := FALSE;
		IF In_Cycle = TRUE THEN
			iStatus:= 1;
		ELSE
			iStatus:=0;	
		END_IF
	END_IF



10: //IF DC Out of Sync
	EnableAxisControl:= FALSE;
	EtherCAT_Master.xRestart := TRUE;
	EtherCAT_Master();
	TimerRecover(PT:=tWait, IN:=TRUE);
	IF TimerRecover.Q=TRUE THEN
		TimerRecover(IN:=FALSE,PT:=T#0S);
		iStatus:=11;
	END_IF
	
11: //Re Initialize Drive
	Restart_Axis(Axis:=AxisVar, bExecute:= TRUE);
	IF Restart_Axis.bDone THEN
		Restart_Axis(Axis:=X, bExecute:= FALSE);
		g_LostSync := FALSE;
		g_FirstSync := FALSE;
		iStatus := -2;
	END_IF
	

		
END_CASE;
AxisControl(Axis:=AxisVar, Enable:=EnableAxisControl);
ActualPosition:=AxisControl.Actual_Position;

HMI_ActualPosition := LREAL_TO_INT(ActualPosition * 1000);

END_FUNCTION_BLOCK

// Recovery
PROGRAM Recovery
VAR
	TimerRecover : TON;
	Restart_X : SMC3_ReinitDrive;
	Restart_Y : SMC3_ReinitDrive;
	Restart_Z : SMC3_ReinitDrive;
	Restart_A : SMC3_ReinitDrive;
	iStatus : INT := -1;
	InRecovery : BOOL := FALSE;
	Done : BOOL := FALSE;
	tWait : TIME := T#5S;
END_VAR

CASE iStatus OF
-1:	//Wait for FirstSync
	IF EtherCAT_Master.xDistributedClockInSync AND  g_FirstSync THEN
		iStatus := 0;
	END_IF
0: // Wait for LostSync
	IF g_LostSync THEN
		iStatus := 10;
		InRecovery := TRUE;
		Done := FALSE;
		gSyncErrors := gSyncErrors + 1;
	END_IF

10: //IF DC Out of Sync
	//dcWindow := DINT_TO_WORD(MaxTotalSyncBufferAvg + 5);
	iStatus:=iStatus+1;

11:	//Restart EtherCAT Master
	EtherCAT_Master.xRestart := TRUE;
	EtherCAT_Master();
	TimerRecover(PT:=tWait, IN:=TRUE);
	IF TimerRecover.Q=TRUE THEN
		TimerRecover(IN:=FALSE,PT:=T#0S);
		iStatus:=iStatus+1;
	END_IF
	
12: //Re Initialize X
	Restart_X(Axis:=X, bExecute:= TRUE);
	IF Restart_X.bDone THEN
		Restart_X(Axis:=X, bExecute:= FALSE);
		iStatus := iStatus+1;
	END_IF

13: //Re Initialize Y
	Restart_Y(Axis:=Y, bExecute:= TRUE);
	IF Restart_Y.bDone THEN
		Restart_Y(Axis:=Y, bExecute:= FALSE);
		iStatus := iStatus+1;
	END_IF
	
14: //Re Initialize Z
	Restart_Z(Axis:=Z, bExecute:= TRUE);
	IF Restart_Z.bDone THEN
		Restart_Z(Axis:=Z, bExecute:= FALSE);
		iStatus := 16;
	END_IF
	
{*  ***Cannot ReInitialize Virtual Drives	
15: //Re Initialize A
	Restart_A(Axis:=A, bExecute:= TRUE);
	IF Restart_A.bDone THEN
		Restart_A(Axis:=A, bExecute:= FALSE);
		iStatus := iStatus+1;
	END_IF
*}
16:	//Finish and Clean Up Recovery
	g_LostSync := FALSE;
	g_FirstSync := FALSE;
	iStatus := -1;
	InRecovery := FALSE;
	Done := TRUE;
	
END_CASE;

END_PROGRAM

// IO_AxisControl
FUNCTION_BLOCK IO_AxisControl
VAR_IN_OUT
	Axis: AXIS_REF_SM3;
END_VAR
VAR_INPUT
	Enable : Bool;
END_VAR
VAR_OUTPUT
	Ready: BOOL;
	Actual_Position: LREAL;
	Actual_Velocity: LREAL;
	Actual_Torque: LREAL;
	AxisError: BOOL;
	AxisErrorID: DWORD;
	Axis_Disabled: BOOL;
	Axis_ErrorStop: BOOL;
	Axis_Stopping: BOOL;
	Axis_Standstill: BOOL;
	Axis_Moving: BOOL;
	Axis_Homing: BOOL;
	Axis_ConstantVelocity: BOOL;
	Axis_Accelerating: BOOL;
	Axis_Decelerating: BOOL;
	Axis_FBError: BOOL;
	Axis_FBErrorID: SMC_ERROR;
	Axis_FBErrorString: STRING(100);
END_VAR
VAR
	Reset: MC_Reset;
	Jog: MC_Jog;
	Power: MC_Power;
	Halt: MC_Halt;
	SetPosition: MC_SetPosition;
	ReadTorque: MC_ReadActualTorque;
	readVelocity: MC_ReadActualVelocity;
	ReadPosition: MC_ReadActualPosition;
	ReadAxisError: mc_ReadaxisError;
	
	ReadStatus: MC_ReadStatus;
	Read_FBError: SMC_ReadFBError;
	GoHome: MC_Home;
END_VAR
VAR // added by the converter: edge detectors and wires of the graphical bodies
    _w1, _w2, _w3, _w4, _w5, _w10, _w12, _w13, _w14, _w16, _w17, _w19, _w20, _w21, _w22, _w23, _w25, _w26, _w27, _w28 : ANY;
    _w6, _w7, _w8, _w9, _w11, _w15, _w18, _w24 : BOOL;
END_VAR

